FUNCTION Convert_USINT_TO_STRING : Hresult
VAR_INPUT
	in : USINT;
	out : REFERENCE TO STRING;
END_VAR
VAR
	converted : STRING;
END_VAR
VAR CONSTANT
	INCOMPATIBLE : HRESULT := 16#9811070E;
END_VAR

converted := USINT_TO_STRING(in);

IF (STRING_TO_USINT(converted) <> in) THEN
	Convert_USINT_TO_STRING := INCOMPATIBLE;
	RETURN;
END_IF

out := converted;

END_FUNCTION

(* stored: Version 1.1.0.1, ProductVersion 3.1.4024.12
   POU Convert_USINT_TO_STRING: Id {5ad3f052-a413-481b-9660-c3c0ffa8b676}, SpecialFunc None *)
